{attribute addProperty BoxType "EJ4002-0000-0018"}
{attribute addProperty Id "Analog_outputAT %Q*INT162"}
{attribute addProperty CRC "4118783225"}
{attribute addProperty SizeInBites "16"}
{attribute addProperty SizeInBytes "2"}
TYPE AO_Output_Channel_F57FA4F9 :
STRUCT
	{attribute addProperty Name "Analog_output"}
	Analog_output AT %Q* : INT;
END_STRUCT
END_TYPE

(* stored: Version 1.2.0.0, ProductVersion 3.1.4024.9
   DUT AO_Output_Channel_F57FA4F9: Id {b6f6843c-c186-49b2-8fbf-3df485cfe8be} *)
